{attribute 'pack_mode' := '1'}
TYPE ST_AddStationSingleDataOut :
STRUCT
	// Fixed data for all methods
	nNumberOfOutputArguments	: UDINT;								// determined amount of output parameters
	nReserved					: ARRAY[1..4] OF BYTE;					// Reserved padding
	
	// Method specific data
	stOutputArgInfo				: ARRAY[1..2] OF ST_UAMethodArgInfo; 	// 
	eStatus						: E_MMServerStatus;						// Status from remote method (succes/fail)
	sMessage					: STRING;								// Debugging message

END_STRUCT
END_TYPE

(* stored: Version 1.1.0.1, ProductVersion 3.1.4024.5
   DUT ST_AddStationSingleDataOut: Id {37c5d574-6cf5-47cd-9671-fa3f4ff51003} *)
